{attribute 'GeneratedUsingTerminal: EL5101--0000'}
{attribute addProperty BoxType "EL5101--0000"}
{attribute addProperty Description "EL5101 1Ch. Encoder 5V"}
{attribute addProperty Physics "KK"}
{attribute addProperty Id "Channel_1AT %I*Channel_B90637B95Channel_1_1AT %Q*Channel_C6781B153WcStateAT %I*WcState_9091E0EB2InfoDataAT %I*InfoData_32EB74EA10"}
{attribute addProperty CRC "310245873"}
{attribute addProperty Size "20"}
TYPE EL5101_127DF9F1 EXTENDS EtcSlaveTerminalBase_947E5A46 :
STRUCT
	{attribute addProperty Name "Channel_1"}
	Channel_1 : Channel_B90637B9;
	{attribute addProperty Name "Channel_1_1"}
	Channel_1_1 : Channel_C6781B15;
	{attribute addProperty Name "WcState"}
	WcState : WcState_9091E0EB;
	{attribute addProperty Name "InfoData"}
	InfoData : InfoData_32EB74EA;
END_STRUCT
END_TYPE

(* stored: Version 1.2.0.0, ProductVersion 3.1.4024.9
   DUT EL5101_127DF9F1: Id {69dc4719-7154-4f05-9e34-9b91da1a1ff0} *)
